// TIA Portal V16 export
// export: Created 2021-04-19T19:30:26.8536143Z, ExportSetting WithDefaults, DisplayName Totally Integrated Automation Portal, DisplayVersion V16 Update 2, DisplayName TIA Portal Version Control Interface, DisplayVersion V16 Update 2, DisplayName TIA Portal Openness, DisplayVersion V16 Update 2, DisplayName STEP 7 Professional, DisplayVersion V16 Update 2, DisplayName STEP 7 Safety, DisplayVersion V16, DisplayName WinCC Advanced, DisplayVersion V16 Update 2
FUNCTION_BLOCK "FB1"   // FB1, FBD
{ S7_Optimized_Access := 'TRUE' }
VERSION : 0.1
// stored: AutoNumber true, IsIECCheckEnabled false, IsRetainMemResEnabled false, MemoryReserve 100, SetENOAutomatically false, UDAEnableTagReadback false
   VAR_INPUT
      IN1 : Bool;
      IN2 : Bool;
   END_VAR
   VAR_OUTPUT
      OUT1 : Bool;
   END_VAR
   VAR_IN_OUT
      INOUT1 : Bool;
   END_VAR
BEGIN

REGION Network 1
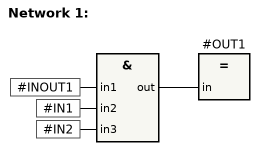
   #OUT1 := #INOUT1 AND #IN1 AND #IN2;
END_REGION
END_FUNCTION_BLOCK
